TYPE "PPrg_Data"
VERSION : 0.1
// Block: PPrg_Data
   STRUCT
      Header : Prg_Header;
   END_STRUCT;

END_TYPE
